TYPE Range2D :
STRUCT
	X : Range;
	Y : Range;
END_STRUCT
END_TYPE

(* stored: Version 1.1.0.1
   DUT Range2D: Id {80f0f29c-5915-0041-1e70-1e15ee0a65af} *)
